FUNCTION SwapNums : INT
VAR_IN_OUT
nNumber3 : INT ;
nNumber4 : INT ;
	
END_VAR
VAR
	nNumberTemp : INT;
	
END_VAR


nNumberTemp := nNumber3;
nNumber3 := nNumber4;
nNumber4 := nNumberTemp;

END_FUNCTION

(* stored: Version 1.1.0.1, ProductVersion 3.1.4024.9
   POU SwapNums: Id {4dd84931-a243-4419-a090-1491cbb4a425}, SpecialFunc None *)
